// TwinCAT 3 PLC project Crane_Control
// ProgramVersion: 3.1.4026.20
// libraries:
//   Tc2_Standard, * (Beckhoff Automation GmbH)
//   Tc2_System, * (Beckhoff Automation GmbH)
// project tree:
//   Enumeration/ E_Mode.TcDUT, E_Motion.TcDUT
//   Function Blocks/ FB_AutoClock.TcPOU (not stored), FB_ControlSignal.TcPOU (not stored), FB_Derivator.TcPOU, FB_FeedForward.TcPOU, FB_FeedForward_NonLinear.TcPOU, FB_Filtering.TcPOU (not stored), FB_Home.TcPOU (not stored), FB_InitialPos.TcPOU (not stored), FB_Integrator.TcPOU (not stored), FB_JoystickInputScaling.TcPOU (not stored), FB_KvFF.TcPOU, FB_MotionRef.TcPOU (not stored), FB_NaiveFF.TcPOU (not stored), FB_Normalize.TcPOU, FB_PID.TcPOU (not stored), FB_PositionInputScaling.TcPOU, FB_PressureFeedback.TcPOU (not stored), FB_RunClock.TcPOU, FB_Running.TcPOU (not stored), FB_ValveOutput.TcPOU
//   Global Variable Lists/ G_Enables.TcGVL (not stored), G_FilterConstants.TcGVL, G_Filtered.TcGVL, G_Init.TcGVL (not stored), G_Inputs.TcGVL, G_Mode.TcGVL, G_OPC.TcGVL, G_Output.TcGVL (not stored), G_Parameter.TcGVL
//   / PlcTask.TcTTO (not stored)
//   Programs/ MAIN.TcPOU (not stored), P_ControlBlock.TcPOU (not stored), P_FeedForward.TcPOU (not stored), P_Filtering.TcPOU (not stored), P_Inputs.TcPOU, P_Modes.TcPOU (not stored), P_Output.TcPOU (not stored), P_PID.TcPOU, P_RunClock.TcPOU

// ---- Enumeration/E_Mode.TcDUT
{attribute 'qualified_only'} // Variable needs to be used with ENUM name
{attribute 'strict'} // Strict rules, prevents invalid assignments/mathematical operations on the ENUM

TYPE E_Mode : // List of settings the program can use, different modes
(
	Off := 0,
	Auto := 1,
	Manuel := 2
);
END_TYPE

// ---- Enumeration/E_Motion.TcDUT
{attribute 'qualified_only'} // Variable needs to be used with ENUM name
{attribute 'strict'} // Strict rules, prevents invalid assignments/mathematical operations on the ENUM
{attribute 'to_string'} // Converts variable into text, to show variable name

TYPE E_Motion : // List of settings the program can use, reference trajectory for motion
(
	Sine,
	Ramp
);
END_TYPE

// ---- Global Variable Lists/G_FilterConstants.TcGVL
{attribute 'qualified_only'}
// LREAL: Long Real decimal number

VAR_GLOBAL
	// Filter constants
	fPressureFilterNum :LREAL := 0.003137;
	fPressureFilterDenz : LREAL := 1.0;
	fPressureFilterDen : LREAL := -0.9969;
	fPressureFilterInit : LREAL := 0.0;
	
	fSignalFilterNum : LREAL := 0.09516;
	fSignalFilterDenz : LREAL := 1.0;
	fSignalFilterDen : LREAL := -0.9048;
	fSignalFilterInit : LREAL := 0.0;
	
	fDerivatorFilterNum : LREAL := 0.0009995;
	fDerivatorFilterDenz : LREAL := 1.0;
	fDerivatorFilterDen : LREAL := -0.999;
	fDerivatorFilterInit : LREAL := 0.0;	
END_VAR

// ---- Global Variable Lists/G_Filtered.TcGVL
{attribute 'qualified_only'}
// LREAL: Long Real decimal number

VAR_GLOBAL
	fPressureSupplyFiltered		: LREAL; // Filtered supply pressure
	fPressurePistonSideFiltered : LREAL; // Filtered pressure, piston side
	fPressureRodSideFiltered 	: LREAL; // Filtered pressure, rod side
	fValveOutputFiltered		: LREAL; // Filtered valve output
	fValveOutputUnfiltered		: LREAL; // Unfiltered valve output
END_VAR

// ---- Global Variable Lists/G_Inputs.TcGVL
{attribute 'qualified_only'} // Variable needs to be used with GVL-name

// INT: [-32768, 32767]	
// BOOL: True/False
// %I* assigns next available memory adress in Twincat (In)

VAR_GLOBAL
	// Mode Selection
	bManual 			AT %I* : BOOL; 	// Manual mode controller
	bAuto	 			AT %I* : BOOL;	// Auto mode controller
	bStartButton		AT %I* : BOOL; 	// Start button
	bStopButton			AT %I* : BOOL;	// Stop button
	
	// Raw Pressure Values
	nRawPa 				AT %I*	: INT;	// Pressure cap side
	nRawPb				AT %I*	: INT;	// Pressure rod side
	nRawPs				AT %I*	: INT;	// Pressure supply
	nRawPaLower			AT %I* 	: INT;	// Pressure under counterbalance valve
	
	// Raw Position Values
	nRawPistonPosition 	AT %I*	: INT;	// Piston position
	nRawJoystick		AT %I*	: INT;	// Joystick Y-position
	nRawFlowSensor		AT %I*	: INT;	// Flow sensor
	nRawSpoolPosition	AT %I*	: INT;	// Spool position
END_VAR

// ---- Global Variable Lists/G_Mode.TcGVL
{attribute 'qualified_only'}
// BOOL: True/False

VAR_GLOBAL // Different modes true/false
	bRunning : BOOL;
	bManual : BOOL;
	bAuto : BOOL;
END_VAR

// ---- Global Variable Lists/G_OPC.TcGVL
{attribute 'qualified_only'}
// LREAL: Long Real decimal number

VAR_GLOBAL
	
	// Unfiltered Pressures
	fPa 				: LREAL; // [bar], Pressure A 
	fPb 				: LREAL; // [bar], Pressure B 
	fPs 				: LREAL; // [bar], Pressure Supply 
	fPaLower 			: LREAL; // [bar], Pressure A between DCV and CBV 
	
	// Filtered Pressures
	fPaFiltered 		: LREAL; // [bar], Pressure A Filtered 
	fPbFiltered 		: LREAL; // [bar], Pressure B Filtered
	fPsFiltered 		: LREAL; // [bar], Pressure Supply Filtered
	fPaLowerFiltered 	: LREAL; // [bar], Pressure A between DCV and CBV Filtered
	
	fSpoolPosition 		: LREAL; // [-1,1], Spool position
	fPistonPosition 	: LREAL; // [m], Piston position
	fPistonPosMeasured 	: LREAL; // [m], Measured piston position
	fJoystick 			: LREAL; // [-1,1], Joystick signal
	fFlow 				: LREAL; // [L/min], Flow rod-side 
	fFlowCalc 			: LREAL; // [L/min], Calculated flow
	
	fXRef 				: LREAL; // [m], Position reference [m]
	fXDotRef 			: LREAL; // [m/s], Velocity reference [m/s]
	fFlowRef 			: LREAL; // [L/min], Flow reference calculated form fXDotRef
	
	fFFFlow				: LREAL; // [L/min], Flow form feed forward
	fKv					: LREAL; // [L/min / bar^0.5] K value 

	fWantedSpoolPos 	: LREAL; // [-1,1], Wanted spool position
	fUpfbGrad 			: LREAL; // Pressure feedback gradient
	fPxGrad 			: LREAL; // Pressure gradient
	fUTest 				: LREAL; // [-1,1], Signal to Valve with pfb (pressure feedback)
	fTime 				: LREAL; // [s], Time
	fError 				: LREAL; // [m], Error
	
	
	fSignalPID 			: LREAL; // PID signal value
	fFF 				: LREAL; // FF signal Value
	fUpfb 				: LREAL; // Pressure feedback signal
	fU 					: LREAL; // [-1,1], Signal to set spool at wanted position 

END_VAR

// ---- Global Variable Lists/G_Parameter.TcGVL
{attribute 'qualified_only'}
// LREAL: Long Real decimal number
// INT: [-32768, 32767]	

VAR_GLOBAL
	// Motion Ref
	// Sine Parameters
	fAmplitude 		: LREAL := 0.15;
	fMean 			: LREAL := 0.2;
	fFrequency 		: LREAL := 0.05;
	
	
	// Valve Values
	// Flow
	fQMaxDown 		: LREAL := 10.0; // [L/min]
	fQMaxUp 		: LREAL := 10.0; // [L/min]	
	
	// Area
	fAreaUp 		: LREAL := 33.100/1E4; //[m^2]
	fAreaDown 		: LREAL := 23.560/1E4; //[m^2]
	
	// Deadband
	fDeadUp 		: LREAL := 0.23;
	fDeadDown 		: LREAL := 0.215;
	
	fMaxSpeed 		: LREAL := 0.01; // [m/s] 
	fDeltaP0 		: LREAL := 8.0; // [Bar]
	
	// Deadband test
	fConst 			: LREAL := 0.0; // [-1, 1]

	fCycleTime 		: LREAL := 0.001; // Time Step [s]. To transfer PLS ticks into real time
	fQConst 		: LREAL := 15;
	fPistonStroke 	: LREAL := 0.5;
	
	// PID-constants
	Kp 				: LREAL := 14.0; 	// P
	Ki 				: LREAL := 0.0;		// I
	Kd 				: LREAL := 0.0;		// D
	
	// Pressure feedback constants
	Kf				: LREAL := 2E-4;
	TauF			: LREAL := 0.1; // [0.05 .. 0.1]
	PFBstate		: INT 	:= 2; // 0:Switching, 1: Pa-phi*Pb, 2: Pb
	FFMode			: INT 	:= 1; // 0: Bachelor FF, 1: Kv FF, 2: Naive FF

END_VAR

// ---- Function Blocks/FB_Derivator.TcPOU
FUNCTION_BLOCK FB_Derivator
// SINT: Integer [-128, 127]
// LREAL: Long Real decimal number

// Constant variables
VAR CONSTANT
	f_SampleRate: LREAL := 1000.0;
END_VAR

// Input variables
VAR_INPUT
	ssMethodType: SINT; // Derivation mode (initialize or next step)
	fSignal: LREAL;		// Signal value to derivate
END_VAR

// Output variables
VAR_OUTPUT
	fSignalDerivative: LREAL; // Output variable after derivation
END_VAR

// Variables
VAR
	rtb_TSamp: LREAL; // run-time-block. Scaled value for time, converts changes per PLC-loop to per second.
	UD_DSTATE: LREAL; // Unit Delay. Current value/internal memory
END_VAR

// Discrete derivation

CASE ssMethodType OF
    SS_INITIALIZE: 
        UD_DSTATE := 0.0; // Reset derivatior
		
    SS_STEP: 
        rtb_TSamp := fSignal * f_SampleRate; // Converts PLC-time into real time. PlcTask cycle tick = 1ms
        fSignalDerivative := rtb_TSamp - UD_DSTATE; // Change of value. Signal this cycle - signal cycle before 
        UD_DSTATE := rtb_TSamp; // Updates current value
END_CASE;

END_FUNCTION_BLOCK

// ---- Function Blocks/FB_FeedForward.TcPOU
FUNCTION_BLOCK FB_FeedForward
// LREAL: Long Real decimal number

// Input variables
VAR_INPUT
	fXDotRef 		: LREAL; // Velocity Reference [m/s]
	fMaxFlowUp 		: LREAL; // Needs to be positive (22)
	fMaxFlowDown 	: LREAL; // Needs to be positive (15)
	fDeadUp			: LREAL; // Needs to be positive (0.155)
	fDeadDown 		: LREAL; // Needs to be positive (0.18)
	
	fPs 			: LREAL; // [Bar]
	fPa 			: LREAL; // [Bar]
	fPb 			: LREAL; // [Bar]
	fDeltaP0		: LREAL; // [Bar] (8.0)
	fAreaUp			: LREAL; // [mm^2]
	fAreaDown		: LREAL; // [mm^2]
END_VAR

// Output variables
VAR_OUTPUT
	fUFF 			: LREAL;	// FF signal value
	fFlow			: LREAL; 	// Wanted Flow
	fFlowLM			: LREAL;	// Flow [L/min]
END_VAR

// Variables
VAR
	fDeltaP_Norm	: LREAL; 	// Pressure Drop with Compensator
	
	fDeltaP			: LREAL; 	// Pressure Drop
	fDeltaP_Ref		: LREAL; 	// Reference Pressure Drop
	fFlowRef		: LREAL; 	// Reference Flow
	
	fUFFTemp		: LREAL;	// Temp Signal Out
END_VAR


fDeltaP_Norm	:= fDeltaP0 * 100000.0; // Converts from Pa

IF fXDotRef > 0.0 THEN // Velocity reference > 0
	fFlow := fXDotRef * fAreaUp; // Calculates wanted flow (Q = v*A)
	fFlowLM := -fFlow * 60000; // Converts flow to [L/min]. Negative sign for valve direction
	fDeltaP := (fPs - fPa) * 100000.0; // Calculates pressure drop
	
	IF fDeltaP < 100 THEN // Safety for pressure drop to never go below 100. Avoiding division by zero
		fDeltaP := 100;
	ELSE
		fDeltaP := fDeltaP;
	END_IF
	
	fDeltaP_Ref := ABS(fDeltaP_Norm/ (fDeltaP)); // Calculates reference pressure drop. 
	fFlowRef := (fFlow * SQRT(fDeltaP_Ref)) * 60000.0; // Calculates reference flow
	fUFFTemp := fFlowRef/fMaxFlowUp; // Normalizes output signal [0,1]
	fUFFTemp := -fUFFTemp * (1.0-fDeadUp); // Adjusts for valve deadband 
	
ELSIF fXDotRef < 0.0 THEN // Velocity reference < 0
	fFlow := fXDotRef * fAreaDown; // Calculates wanted flow (Q = v*A)
	fFlowLM := -fFlow * 60000; // Converts flow to [L/min]. Negative sign for valve direction
	fDeltaP := (fPs - fPb) * 100000.0; // Calculates pressure drop
	
	IF fDeltaP < 100 THEN // Safety for pressure drop to never go below 100. Avoiding division by zero
		fDeltaP := 100;
	ELSE
		fDeltaP := fDeltaP;
	END_IF
	
	fDeltaP_Ref := ABS(fDeltaP_Norm/(fDeltaP)); // Calculates reference pressure drop
	fFlowRef := (fFlow * SQRT(fDeltaP_Ref)) * 60000.0; // Calculates reference flow
	fUFFTemp := fFlowRef/fMaxFlowDown; // Normalizes output signal [-1,0]
	fUFFTemp := -fUFFTemp*(1.0-fDeadDown); // Adjusts for valve deadband
	
ELSE
	
	fUFFTemp := 0.0; // FF signal is zero		

END_IF

// Safety to keep FF signal [-1,1]
IF fUFFTemp > 1.0 THEN
	fUFF := 1.0;
ELSIF fUFFTemp < -1.0 THEN
	fUFF := -1.0;
ELSE
	fUFF := fUFFTemp;
END_IF

END_FUNCTION_BLOCK

// ---- Function Blocks/FB_FeedForward_NonLinear.TcPOU
FUNCTION_BLOCK FB_FeedForward_NonLinear
// LREAL: Long Real decimal number

// Input variables
VAR_INPUT
	fXDotRef 		: LREAL; // Velocity Reference [m/s]
	fMaxFlowUp 		: LREAL; // Needs to be positive (22)
	fMaxFlowDown 	: LREAL; // Needs to be positive (15)
	fDeadUp			: LREAL; // Needs to be positive (0.155)
	fDeadDown 		: LREAL; // Needs to be positive (0.18)

	fPs 			: LREAL; // [Bar]
	fPa 			: LREAL; // [Bar]	
	fPb 			: LREAL; // [Bar]
	fDeltaP0		: LREAL; // [Bar]
	fAreaUp			: LREAL; // [mm^2]
	fAreaDown		: LREAL; // [mm^2]
END_VAR

// Output variables
VAR_OUTPUT
	fUFF 			: LREAL;	// FF signal value
	fFlow			: LREAL; 	// Wanted Flow
	fFlowLM			: LREAL;	// Flow [L/min]
END_VAR

// Variables
VAR
	fDeltaP_Norm	: LREAL; 	// Pressure Drop with Compensator
	
	fDeltaP			: LREAL; 	// Pressure Drop
	fDeltaP_Ref		: LREAL; 	// Reference Pressure Drop
	fFlowRef		: LREAL; 	// Reference Flow
	
	fUFFTemp		: LREAL;	// Temp Signal Out
END_VAR

// Non-linear FF compensates for disturbances where the relationship is not proportional/constant. 

fDeltaP_Norm	:= fDeltaP0 * 100000.0; // Converts to Pa

IF fXDotRef > 0.0 THEN // Velocity reference > 0
	
	fFlow := fXDotRef * fAreaUp; // Calculates wanted flow 
	fFlowLM := -fFlow * 60000; // Converts flow to [L/min]. Negative sign for valve direction
	fDeltaP := (fPs - fPa) * 100000.0; // Calculates pressure drop
	IF fDeltaP < 100 THEN // Safety for pressure drop to never go below 100. Avoiding division by zero
		fDeltaP := 100;
	ELSE
		fDeltaP := fDeltaP;
	END_IF
	fDeltaP_Ref := ABS(fDeltaP_Norm/ (fDeltaP)); // Calculates reference pressure drop
	fFlowRef := (fFlow * SQRT(fDeltaP_Ref)) * 60000.0; // Calculates reference flow
	fUFFTemp := fFlowRef/fMaxFlowUp; // Normalizes output signal [0,1]
	fUFFTemp := -fUFFTemp * (1.0-fDeadUp); // Adjusts for valve deadband
	
ELSIF fXDotRef < 0.0 THEN // Velocity reference < 0
	
	fFlow := fXDotRef * fAreaDown; // Calculates wanted flow 
	fFlowLM := -fFlow * 60000; // Converts flow to [L/min]. Negative sign for valve direction
	fDeltaP := (fPs - fPb) * 100000.0; // Calculates pressure drop
	
	IF fDeltaP < 100 THEN // Safety for pressure drop to never go below 100. Avoiding division by zero
		fDeltaP := 100; 
	ELSE
		fDeltaP := fDeltaP; 
	END_IF
	
	fDeltaP_Ref := ABS(fDeltaP_Norm/(fDeltaP)); // Calculates reference pressure drop
	fFlowRef := (fFlow * SQRT(fDeltaP_Ref)) * 60000.0; // Calculates reference flow
	fUFFTemp := fFlowRef/fMaxFlowDown; // Normalizes output signal [0,1]
	fUFFTemp := -fUFFTemp*(1.0-fDeadDown); // Adjusts for valve deadband
	
ELSE
	
	fUFFTemp := 0.0;		

END_IF

// Safety to keep FF signal [-1,1]
IF fUFFTemp > 1.0 THEN
	fUFF := 1.0;
ELSIF fUFFTemp < -1.0 THEN
	fUFF := -1.0;
ELSE
	fUFF := fUFFTemp;
END_IF

END_FUNCTION_BLOCK

// ---- Function Blocks/FB_KvFF.TcPOU
FUNCTION_BLOCK FB_KvFF
// LREAL: Long Real decimal number

// Input variables
VAR_INPUT
	fPs 		: LREAL; // [bar] 
	fPa 		: LREAL; // [bar]
	fPb 		: LREAL; // [bar]
	fXDotRef 	: LREAL; // [m/s]
END_VAR

// Output variables
VAR_OUTPUT
	fFFTemp		: LREAL; // [-1,1], Wanted spool position
	fFF 		: LREAL; // [-1,1], Spool signal for position
	fFlow 		: LREAL; // [L/min]
	fKv 		: LREAL; // [L/min / bar^0.5]
END_VAR

// Variables
VAR
	fDeltaP		: LREAL; // [bar]
END_VAR



IF fXDotRef > 0.0 THEN // Velocity reference > 0
	IF fKv >= 0.1 THEN 
		fFFTemp := -0.013*EXPT(fKv,5) + 0.1355*EXPT(fKv,4) - 0.5012*EXPT(fKv,3) + 0.7175*EXPT(fKv,2) - 0.0278 * fKv + 0.2684; // Curve fitting for valve opening
	ELSIF fKv < 0.1 THEN
		fFFTemp := 0.2325 + 0.0398 * fKv/0.1; // Linear approximation for low Kv values
	ELSE 
		fFFTemp := G_Parameter.fDeadUp; // Fallback to deadband value (positive direction)
	END_IF
	fFlow := fXDotRef * G_Parameter.fAreaUp * 6E4; // Calculates flow
	fDeltaP := fPs - fPa; // Calculates pressure drop
	fFF := -(fFFTemp + 0.0151)/1.1224; // Scaling and offset
	
ELSIF fXDotRef < 0.0 THEN // Velocity reference < 0
	IF fKv >= 0.1 THEN
		fFFTemp := 0.0054*EXPT(fKv,6) - 0.0733*EXPT(fKv,5) + 0.3796*EXPT(fKv,4) - 0.9356*EXPT(fKv,3) + 1.0359*EXPT(fKv,2) - 0.1046 * fKv + 0.2381; // Curve fitting for valve opening
	ELSIF fKv < 0.1 THEN
		fFFTemp := 0.2175 + 0.0196 * fKv/0.1; // Linear approximation for low Kv values
	ELSE 
		fFFTemp := G_Parameter.fDeadDown; // Fallback to deadband value (negative direction)
	END_IF
	fFlow := fXDotRef * G_Parameter.fAreaDown * 6E4; // Calculates flow
	fDeltaP := fPs - fPb; // Calculates pressure drop
	fFF := (fFFTemp + 0.0398)/1.1079; // Scaling and offset
	
ELSE
	fFlow := 0.0;
	fFFTemp := 0.0;
	fFF := 0.0;
END_IF

// Safety to avoid division by zero when pressure drop is below 0
IF fDeltaP <= 0.0 THEN
	fKv := 4.0;
ELSE
	fKv := ABS(fFlow)/SQRT(fDeltaP);
END_IF

END_FUNCTION_BLOCK

// ---- Function Blocks/FB_Normalize.TcPOU
FUNCTION_BLOCK FB_Normalize
// INT: [-32768, 32767]	
// LREAL: Long Real decimal number

// Constant variables
VAR CONSTANT
	MaxBitValue : LREAL := 32767.0;
END_VAR

// Input variables
VAR_INPUT
	nRawInput : INT;
	fMaxValue : LREAL;
END_VAR

// Output variables
VAR_OUTPUT
	fNormalizedInput : LREAL;
END_VAR

fNormalizedInput := (fMaxValue	* INT_TO_LREAL(nRawInput)) / MaxBitValue;
// Value/Max-value = Raw_value/Max-raw_value. Uses this definition to calculate value for normalized data.
// Int_to_Lreal makes an integer into a long real decimal number
// 16 bit = [-32767, 32767], max value: 32 767

fNormalizedInput := LIMIT(0, fNormalizedInput, fMaxValue); // Limit(min, test-value, max)
// Safety function. Lowest value = 0, highest = f_MaxValue

END_FUNCTION_BLOCK

// ---- Function Blocks/FB_PositionInputScaling.TcPOU
FUNCTION_BLOCK FB_PositionInputScaling
// LREAL: Long Real decimal number
// INT: [-32768, 32767]

// Input variables
VAR_INPUT
	nRawInput 				: INT; // Raw position
	fMaxInputValue 			: LREAL; 
	fMinInputValue			: LREAL;
	fMaxOutputValue  		: LREAL;
	fMinOutputValue  		: LREAL;	
END_VAR

// Output variables
VAR_OUTPUT
	fOutput : LREAL;
	fActual : LREAL;
END_VAR

// Variables
VAR
	fRawInput : LREAL;
	fNormalizedInput: LREAL;
	fTempOut : LREAL; // Temporary output
END_VAR

fRawInput := INT_TO_LREAL(nRawInput); // Converts into a decimal number

fNormalizedInput := (fRawInput - fMinInputValue) / (fMaxInputValue - fMinInputValue); // Normalized input [0,1]
fTempOut := fMinOutputValue + fNormalizedInput*(fMaxOutputValue - fMinOutputValue); // Converts percentage into real value [0, 0.5]

fOutput := LIMIT(fMinOutputValue, fTempOut, fMaxOutputValue); // Safety limit [0, value, 0.5]
fActual := LIMIT(fMinOutputValue, fTempOut - 0.0006 - 0.0109*fTempOut + 0.5855*EXPT(fTempOut,2) - 1.1291*EXPT(fTempOut,3), fMaxOutputValue);
// Curve fitting to remove offsets

END_FUNCTION_BLOCK

// ---- Function Blocks/FB_RunClock.TcPOU
FUNCTION_BLOCK FB_RunClock
// LREAL: Long Real decimal number	
// BOOL: True/False

// Input variables
VAR_INPUT
	bStart 		: BOOL; // Set to true
	bStop 		: BOOL; // Stop button on controller
	fCycleTime  : LREAL; // Time step [s]
END_VAR

// Output variables
VAR_OUTPUT
	fTime : LREAL; // Output (time)
END_VAR

// Variables
VAR
	bOnOff : BOOL; // True/False
END_VAR

IF bStop OR (G_Work.eStatus = E_Status.Off) THEN // If stop button is pressed or system is off 
	bOnOff := FALSE; 
	fTime := 0.0; 
ELSIF bOnOff OR bStart THEN // If system is online/start button pushed, start timer
	bOnOff := TRUE;
	fTime := fTime + fCycleTime;
END_IF

END_FUNCTION_BLOCK

// ---- Function Blocks/FB_ValveOutput.TcPOU
FUNCTION_BLOCK FB_ValveOutput
// LREAL: Long Real decimal number
// INT: [-32768, 32767]	
// BOOL: True/False

// Input variables
VAR_INPUT
	bEnable 			: BOOL; 
	fNormalizedInput 	: LREAL;
END_VAR

// Output variables
VAR_OUTPUT
	nOutput : INT; 
END_VAR

// Variables
VAR
	nOffset 	: LREAL := 19630.0; // Closed valve
	nMaxValue	: LREAL := 29460.0; // Max value valve
	nMinValue 	: LREAL :=  9830.0; // Min value valve
	nTempOutput : LREAL; // Temporary output
END_VAR


IF fNormalizedInput > 0.0 THEN // fNormalizedInput = Signal to set spool at wanted position [-1,1]
	nTempOutput := (fNormalizedInput) * (nMaxValue - nOffset) + nOffset; // Converts wanted signal [-1,1] into <Closed valve, nMaxValve], positive direction
ELSIF fNormalizedInput < 0.0 THEN
	nTempOutput := (fNormalizedInput) * (nOffset - nMinValue) + nOffset; // Converts wanted signal into [nMinValve, Closed valve>, negative direction
ELSE 
	nTempOutput := nOffset; // If wanted spool position = 0, output = closed valve
END_IF


IF NOT(bEnable) THEN // If bEnable is false, close valve
	nOutput := LREAL_TO_INT(nOffset);
ELSIF (bEnable) THEN // Else send output
	nOutput := LREAL_TO_INT(nTempOutput);	
END_IF

END_FUNCTION_BLOCK

// ---- Programs/P_Inputs.TcPOU
PROGRAM P_Inputs
// LREAL: Long Real decimal number

VAR
	fbNormPa :  FB_Normalize;
	fbNormPb :  FB_Normalize;
	fbNormPs :  FB_Normalize;
	fbNormPaLower : FB_Normalize;
	
	fbNormPistonPosition : FB_PositionInputScaling;
	fbNormSpoolPosition : FB_JoystickInputScaling;
	fbJoystick : FB_JoystickInputScaling;	// Hvorfor bruker de joystick input scaling?
	fbFlow	: FB_JoystickInputScaling;		// Samme her^

	fPa : LREAL;
	fPb : LREAL;
	fPs : LREAL;
	fPaLower : LREAL;
	
	fPistonPosition : LREAL;
END_VAR

// Runs FBs with given values

fbNormPa(
	nRawInput := G_Inputs.nRawPa,	// Raw value pressure A
	fMaxValue := 400.0, 			// [Bar]
	fNormalizedInput => G_OPC.fPa	// Unfiltered pressure A out from FB (normalized)
);

fbNormPb(
	nRawInput := G_Inputs.nRawPb,	// Raw value pressure B
	fMaxValue := 400.0, 			// [Bar]
	fNormalizedInput => G_OPC.fPb	// Unfiltered pressure B out from FB (normalized)
);

fbNormPs(
	nRawInput := G_Inputs.nRawPs,	// Raw value pressure S
	fMaxValue := 400.0, 			// [Bar]
	fNormalizedInput => G_OPC.fPs 	// Unfiltered pressure S out from FB (normalized)
);

fbNormPistonPosition(
	nRawInput := G_Inputs.nRawPistonPosition,
	
	fMaxInputValue := 16090.0,
	fMinInputValue := 125.0,
	fMaxOutputValue := 0.5,
	fMinOutputValue := 0.0,	
	
	fOutput => G_OPC.fPistonPosMeasured,
	fActual => G_OPC.fPistonPosition
);
	
fbJoystick(
	nRawInput := G_Inputs.nRawJoystick, // Joystick raw y-position
	fMaxValue := 1.0,
	bEnable := (G_Mode.bRunning AND G_Mode.bManual), // Running and manual needs to be on
	
	fMaxInputValue := 14746.0,
	fMinInputValue := 1617.0,
	fNeutralInputValue := 8160.0,
	fNeutralDeadband := 100.0,
	
	fOutput => G_OPC.fJoystick // Joystick output
);

fbNormPaLower(
	nRawInput := G_Inputs.nRawPaLower, 	// Raw pressure A lower
	fMaxValue := 400.0, 				// [Bar]
	fNormalizedInput => G_OPC.fPaLower	// Unfiltered pressure A lower out from FB (normalized)
);

fbNormSpoolPosition(
	nRawInput := G_Inputs.nRawSpoolPosition,
	fMaxValue := 1.0,
	bEnable := TRUE,
	
	fNeutralInputValue := 8355.0,
	fMaxInputValue := 12645.0,
	fMinInputValue := 4071,
	fNeutralDeadband := 15.0,
	
	fOutput => G_OPC.fSpoolPosition
);

fbFlow(
	bEnable := TRUE,
	nRawInput := G_Inputs.nRawFlowSensor,
	fMaxValue := 150.0, // [l/min]
	
	fMaxInputValue := 32767.0,
	fMinInputValue := 0,
	fNeutralInputValue := 15270.0,
	fNeutralDeadband := 25.0,
	
	fOutput => G_OPC.fFlow
);

END_PROGRAM

// ---- Programs/P_PID.TcPOU
PROGRAM P_PID
VAR
	fbPID : FB_PID;
	fbIntegrator : FB_Integrator;
	fbDerivator : FB_Derivator;
	fbDerivatorFiltering : FB_Filtering;
END_VAR


fbPID(
	fX := G_OPC.fXRef, 					// Position reference
	fXReal := G_OPC.fPistonPosition, 	// Piston position
		
	fError => G_OPC.fError
);

IF (G_Enables.bEnablePID AND G_Mode.bRunning) THEN // PID activated and system running
	
	fbDerivatorFiltering(
		ssMethodType := 1,
		Signal := fbPID.fSignalD,
		Num := G_FilterConstants.fDerivatorFilterNum,
		Denz := G_FilterConstants.fDerivatorFilterDenz,
		Den := G_FilterConstants.fDerivatorFilterDen,
		Initial := G_FilterConstants.fDerivatorFilterInit,
		Signal_Filtered => fbDerivator.fSignal
	);
	
	fbIntegrator(
		ssMethodType := BOOL_TO_SINT(G_Inputs.bStartButton),
		fSignal := fbPID.fSignalI,
		fSignalIntegrated => fbPID.fSignalIntegrated // Sends to PID FB
	);
	fbDerivator(
		ssMethodType := BOOL_TO_SINT(G_Inputs.bStartButton),
		fSignal := fbPID.fSignalD,
		fSignalDerivative => fbPID.fSignalDerivated
	);

	fbPID(
		bEnablePID := G_Enables.bEnablePID,
		fX := G_OPC.fXRef,
		fXReal := G_OPC.fPistonPosition,
		fKp := G_Parameter.Kp,
		fKi := G_Parameter.Ki,
		fKd := G_Parameter.Kd,
		
		fSignalAdjusted => G_OPC.fSignalPID
	);

END_IF

END_PROGRAM

// ---- Programs/P_RunClock.TcPOU
PROGRAM P_RunClock

VAR
	fbRunClock : FB_RunClock; 
END_VAR

// Runs FB with given values
fbRunClock(
	bStart := TRUE,
	bStop := G_Inputs.bStopButton, // Stop button on controller
	fCycleTime := G_Parameter.fCycleTime, // Time step
	
	fTime => G_OPC.fTime // Output time 
);

END_PROGRAM
